INTERFACE I_Filter

METHOD SetFilter : BOOL
VAR_INPUT
	FilterPos	: USINT;
END_VAR
END_METHOD

END_INTERFACE

(* stored: Version 1.1.0.1, ProductVersion 3.1.4024.13
   POU I_Filter: Id {369ce03b-3dae-4f80-85b9-cf8255ffdfa1}, SpecialFunc None
   Method SetFilter: Id {f495802b-4026-4457-9091-482dcab0997f} *)
